Yaskawa INFORM job: R1_W35-36-A2(90,0)KM-OK.JBI

/JOB
//NAME R1_W35-36-A2(90,0)KM-OK
///FOLDERNAME KRIS-SCIANA
//POS
///NPOS 106,106,0,8,0,0
///TOOL 0
///POSTYPE PULSE
///PULSE
C00000=133203,-151163,-123299,-9717,62642,66340
C00001=174797,-117356,-116748,-21269,45538,71767
C00002=167772,-84002,-97078,-14094,48870,67877
C00003=165686,-78458,-91681,-12461,48082,67072
C00004=164380,-75033,-87353,-11529,47009,66627
C00005=163956,-73698,-86723,-11111,47244,66408
C00006=164380,-75033,-87353,-11529,47009,66627
C00007=164380,-75168,-86749,-11611,46576,66681
C00008=164380,-75033,-87353,-11529,47009,66627
C00009=153920,-88304,-92067,12036,39705,58111
C00010=154679,-95974,-98045,11331,39340,58456
C00011=173550,-85466,-94205,-27435,46132,79851
C00012=171230,-80075,-88912,-25751,44973,79042
C00013=169766,-76569,-85027,-24769,44003,78586
C00014=169296,-75333,-84452,-24248,44125,78311
C00015=169766,-76569,-85027,-24769,44003,78586
C00016=169766,-76625,-84526,-24915,43697,78678
C00017=169766,-76569,-85027,-24769,44003,78586
C00018=181492,-65329,-82160,-40061,58474,82712
C00019=194013,-96570,-98942,-47807,60580,87756
C00020=194013,-96570,-98942,-47807,60580,-51245
C00021=203995,-38561,-98383,-32392,87811,-61268
C00022=215531,-14026,-76080,-16989,89427,-64069
C00023=220381,23081,-47382,-28420,104834,-69323
C00024=222470,49341,-20749,-34117,110874,-70142
C00025=221806,39036,-18377,-32558,104968,-68512
C00026=221724,38193,-19154,-32548,104980,-68545
C00027=221793,39711,-18991,-32681,105579,-68702
C00028=221571,37477,-21115,-32657,105643,-68801
C00029=221571,37188,-20943,-32612,105427,-68735
C00030=222926,39369,-21029,-33153,106861,-68698
C00031=223966,38557,-20553,-33262,106600,-68250
C00032=226583,52363,-1545,-40953,111419,-72507
C00033=222365,54755,1299,-40199,109281,-73389
C00034=223739,53056,-5101,-41284,112199,-74042
C00035=218620,27349,-37181,-28911,103712,-69795
C00036=215610,8993,-54476,-21168,96493,-66602
C00037=215610,8993,-54476,-21168,96493,-66602
C00038=181695,45814,-29997,-12378,123903,-78661
C00039=175710,42579,-26967,-11179,119789,-80079
C00040=175710,41251,-26577,-11066,118883,-79984
C00041=175710,40643,-26381,-11016,118459,-79940
C00042=175710,41109,-26532,-11055,118786,-79974
C00043=179718,49925,-16862,-11334,117833,-78596
C00044=179718,48988,-16533,-11255,117161,-78526
C00045=179840,47754,-17901,-11295,117380,-78511
C00046=180929,51970,-15477,-11489,118166,-78244
C00047=186701,44441,-23841,-12245,120091,-76601
C00048=186701,44089,-23732,-12211,119848,-76573
C00049=186701,43441,-23524,-12148,119396,-76521
C00050=186701,43791,-23639,-12182,119641,-76549
C00051=186455,51365,-15254,-11993,118371,-76483
C00052=186455,50629,-14996,-11926,117845,-76424
C00053=186489,49492,-16087,-11940,117934,-76422
C00054=186464,52211,-15044,-12032,118669,-76513
C00055=197498,49366,-18518,-13101,120698,-73153
C00056=197498,48966,-18393,-13058,120422,-73119
C00057=197498,48360,-18192,-12995,119997,-73065
C00058=197498,48957,-18389,-13057,120414,-73118
C00059=196870,57395,-8813,-12787,118814,-73130
C00060=196870,56102,-8342,-12659,117882,-73019
C00061=196979,54648,-10005,-12704,118165,-73017
C00062=197536,59091,-8206,-12907,119386,-72980
C00063=207821,58971,-8346,-13607,120773,-69731
C00064=207821,58374,-8156,-13541,120362,-69677
C00065=207821,57623,-7899,-13459,119832,-69608
C00066=207821,58153,-8083,-13517,120207,-69656
C00067=206745,66427,1648,-13203,118369,-69786
C00068=206745,65417,2036,-13100,117629,-69695
C00069=206913,64191,584,-13146,117909,-69674
C00070=207056,66191,1124,-13250,118607,-69712
C00071=206807,76962,-1437,-14356,125245,-70692
C00072=178606,-7084,-71070,-5513,93657,-76211
C00073=178606,-12434,-69077,-5488,89699,-76039
C00074=178606,-14822,-67880,-5486,87744,-75953
C00075=166292,-14208,-67445,-208,87128,-79433
C00076=169556,-31327,-73894,-6745,74234,-79609
C00077=174833,-45592,-87827,-10016,75291,-78208
C00078=186297,-11008,-70403,4453,90875,-67936
C00079=188919,-9021,-66869,3281,89626,-67272
C00080=188904,-12076,-65397,3288,87157,-67339
C00081=208785,1057,-55100,-5592,87804,-61823
C00082=208466,4683,-57667,-5460,91212,-62059
C00083=165581,-6998,-67341,13530,92866,-73359
C00084=173591,4611,-59645,1891,100899,-73578
C00085=173591,2327,-58796,1879,99203,-73603
C00086=194456,6891,-54971,-5453,99565,-67936
C00087=194382,12631,-57077,-5530,103787,-68146
C00088=175852,-51384,-92394,-10580,75239,-77894
C00089=192163,-96959,-104003,-46570,61456,86648
C00090=152921,-122541,-108068,855,30408,65915
C00091=145454,-97772,-94010,9448,34954,61648
C00092=146863,-93018,-91491,7663,35693,62543
C00093=145492,-97786,-92846,9577,34237,61575
C00094=144929,-94903,-92971,9846,35841,61460
C00095=146748,-90810,-92138,6152,39176,62647
C00096=145438,-91687,-92725,7508,39198,61958
C00097=146922,-92489,-91306,7569,35844,62592
C00098=145432,-97676,-94179,9438,35110,61655
C00099=146808,-105604,-100046,7956,34504,62387
C00100=157428,-158903,-123496,-7044,21383,69853
C00101=121608,-159131,-116680,-7067,21310,69864
C00102=121608,-159131,-116680,-7067,21310,69864
C00103=6794,-159131,-116680,-7067,21310,69864
C00104=-19798,29541,-22378,6716,72357,-39538
C00105=-2234,110189,19387,12809,93315,-86753
BC00000=338018,1185852,1068216
BC00001=322204,1189606,1068222
BC00002=322204,1189606,1068222
BC00003=322204,1189606,1068222
BC00004=322204,1189606,1068222
BC00005=322204,1189606,1068222
BC00006=322204,1189606,1068222
BC00007=322204,1189606,1068222
BC00008=322204,1189606,1068222
BC00009=322204,1189606,1068222
BC00010=322204,1189606,1068222
BC00011=359570,1189606,1068222
BC00012=359570,1189606,1068222
BC00013=359570,1189606,1068222
BC00014=359570,1189606,1068222
BC00015=359570,1189606,1068222
BC00016=359570,1189606,1068222
BC00017=359570,1189606,1068222
BC00018=359570,1189606,1068222
BC00019=359570,1189606,1068222
BC00020=359570,1189606,1068222
BC00021=359570,1189606,1068222
BC00022=359570,1189606,1068222
BC00023=359570,1189606,1068222
BC00024=359570,1189606,1068222
BC00025=359570,1384690,1084352
BC00026=359570,1384690,1084352
BC00027=359570,1384690,1084352
BC00028=359570,1384690,1084352
BC00029=359570,1384690,1084352
BC00030=359570,1384690,1084352
BC00031=359570,1384690,1084352
BC00032=359570,1384690,1084352
BC00033=359570,1384690,1084352
BC00034=359570,1384690,1084352
BC00035=359570,1189606,1068222
BC00036=359570,1189606,1068222
BC00037=359570,1189606,1068222
BC00038=359570,1189606,1068222
BC00039=359570,1189606,1068222
BC00040=359570,1189606,1068222
BC00041=359570,1189606,1068222
BC00042=359570,1189606,1068222
BC00043=359570,1189606,1068222
BC00044=359570,1189606,1068222
BC00045=359570,1189606,1068222
BC00046=359570,1189606,1068222
BC00047=359570,1189606,1068222
BC00048=359570,1189606,1068222
BC00049=359570,1189606,1068222
BC00050=359570,1189606,1068222
BC00051=359570,1189606,1068222
BC00052=359570,1189606,1068222
BC00053=359570,1189606,1068222
BC00054=359570,1189606,1068222
BC00055=359570,1189606,1068222
BC00056=359570,1189606,1068222
BC00057=359570,1189606,1068222
BC00058=359570,1189606,1068222
BC00059=359570,1189606,1068222
BC00060=359570,1189606,1068222
BC00061=359570,1189606,1068222
BC00062=359570,1189606,1068222
BC00063=359570,1189606,1068222
BC00064=359570,1189606,1068222
BC00065=359570,1189606,1068222
BC00066=359570,1189606,1068222
BC00067=359570,1189606,1068222
BC00068=359570,1189606,1068222
BC00069=359570,1189606,1068222
BC00070=359570,1189606,1068222
BC00071=359570,1189606,1068222
BC00072=359570,1189606,1068222
BC00073=359570,1189606,1068222
BC00074=359570,1189606,1068222
BC00075=359570,1189606,1068222
BC00076=359570,1189606,1068222
BC00077=359570,1189606,1068222
BC00078=359570,1189606,1068222
BC00079=359570,1189606,1068222
BC00080=359570,1189606,1068222
BC00081=359570,1189606,1068222
BC00082=359570,1189606,1068222
BC00083=359570,1189606,1068222
BC00084=359570,1189606,1068222
BC00085=359570,1189606,1068222
BC00086=359570,1189606,1068222
BC00087=359570,1189606,1068222
BC00088=359570,1189606,1068222
BC00089=359570,1189606,1068222
BC00090=340811,1189606,1068222
BC00091=340087,1189606,1068222
BC00092=339797,1189606,1068222
BC00093=339797,1189606,1068222
BC00094=339797,1189606,1068222
BC00095=305385,1189606,1068222
BC00096=302058,1189606,1068222
BC00097=290425,1189606,1068222
BC00098=290715,1189606,1068222
BC00099=291439,1189606,1068222
BC00100=291439,1189606,1068222
BC00101=291439,1189606,1068222
BC00102=387760,1226770,1068222
BC00103=387760,1189606,1068222
BC00104=204934,1269644,1068209
BC00105=126121,1277269,1068204
///POSTYPE BASE
///RECTAN
///RCONF 0,0,0,0,0,0,0,0,0,0,0,0,0,0,0,0,0,0,0,0,0,0,0,0
P00006=0.222,-3.123,-1.508,0.0000,0.0000,0.0000
P00021=-0.225,-6.128,-0.405,0.0000,0.0000,0.0000
P00022=0.222,-3.123,-1.508,0.0000,0.0000,0.0000
P00025=-2.003,0.006,0.728,0.0000,0.0000,0.0000
P00030=5.926,-4.294,-1.390,0.0000,0.0000,0.0000
P00031=1.853,-0.001,-1.549,0.0000,0.0000,0.0000
P00032=1.957,0.503,-7.217,0.0000,0.0000,0.0000
///RCONF 0,0,0,0,1,0,0,0,0,0,0,0,0,0,0,0,0,0,0,0,0,0,0,0
P00033=-0.123,0.612,-5.012,0.0000,0.0000,0.0000
//INST
///DATE 2024/07/22 18:40
///ATTR SC,RW
///GROUP1 RB1,BS1
NOP
'r1_W35-36-A2(90,0)
'Path S1033 (for W914)
SFTOF
MOVJ C00000 BC00000 VJ=20.00
MOVJ C00001 BC00001 VJ=20.00
MOVL C00002 BC00002 V=166.7
MOVL C00003 BC00003 V=166.7
MOVL C00004 BC00004 V=60.0
REFP 3 C00005 BC00005
CALL JOB:SEARCH-R1
SET P021 P006
SFTON P021
MOVL C00006 BC00006 V=60.0
REFP 3 C00007 BC00007
CALL JOB:SEARCH-R1
SET P021 P006
SFTON P021
MOVL C00008 BC00008 V=60.0
MOVL C00009 BC00009 V=166.7
MOVL C00010 BC00010 V=166.7
'Path S1034 (for W914)
SFTOF
MOVL C00011 BC00011 V=166.7
MOVL C00012 BC00012 V=166.7
MOVL C00013 BC00013 V=60.0
REFP 3 C00014 BC00014
CALL JOB:SEARCH-R1
SET P022 P006
SFTON P022
MOVL C00015 BC00015 V=60.0
REFP 3 C00016 BC00016
CALL JOB:SEARCH-R1
SET P022 P006
SFTON P022
MOVL C00017 BC00017 V=60.0
MOVL C00018 BC00018 V=166.7
MOVJ C00019 BC00019 VJ=20.00
MOVJ C00020 BC00020 VJ=100.00
MOVJ C00021 BC00021 VJ=100.00
SFTOF
MOVJ C00022 BC00022 VJ=100.00
MOVJ C00023 BC00023 VJ=50.00
MOVJ C00024 BC00024 VJ=60.00
COMM PAUSE
COMM MOVL C00025 BC00025 V=60.0
COMM REFP 3 C00026 BC00026
COMM CALL JOB:SEARCH-R1
COMM SET P025 P006
COMM SFTON P025
COMM MOVL C00027 BC00027 V=83.3
COMM MOVL C00028 BC00028 V=60.0
COMM REFP 3 C00029 BC00029
COMM CALL JOB:SEARCH-R1
COMM SET P025 P006
COMM SFTON P025
COMM MOVL C00030 BC00030 V=60.0
COMM MOVL C00031 BC00031 V=166.7
COMM MACRO1 MJ#(0) ARGF6
COMM SFTON P025
COMM MOVJ C00032 BC00032 VJ=10.00
COMM MOVL C00033 BC00033 V=13.3
COMM ARCOF
COMM MOVL C00034 BC00034 V=83.3
COMM SFTOF
COMM PAUSE
MOVL C00035 BC00035 V=166.7
MOVJ C00036 BC00036 VJ=20.00
MOVL C00037 BC00037 V=166.7
MOVJ C00038 BC00038 VJ=20.00
MOVL C00039 BC00039 V=233.3
MOVL C00040 BC00040 V=60.0
REFP 3 C00041 BC00041
CALL JOB:SEARCH-R1
SET P030 P006
SFTON P030
MOVL C00042 BC00042 V=60.0
MOVL C00043 BC00043 V=100.0
MOVL C00044 BC00044 V=60.0
REFP 3 C00045 BC00045
CALL JOB:SEARCH-R1
SET P030 P006
SFTON P030
MOVL C00046 BC00046 V=60.0
SFTOF
MOVL C00047 BC00047 V=233.3
MOVL C00048 BC00048 V=60.0
REFP 3 C00049 BC00049
CALL JOB:SEARCH-R1
SET P031 P006
SFTON P031
MOVL C00050 BC00050 V=60.0
MOVL C00051 BC00051 V=100.0
MOVL C00052 BC00052 V=60.0
REFP 3 C00053 BC00053
CALL JOB:SEARCH-R1
SET P031 P006
SFTON P031
MOVL C00054 BC00054 V=60.0
SFTOF
MOVL C00055 BC00055 V=233.3
MOVL C00056 BC00056 V=60.0
REFP 3 C00057 BC00057
CALL JOB:SEARCH-R1
SET P032 P006
SFTON P032
MOVL C00058 BC00058 V=60.0
MOVL C00059 BC00059 V=100.0
MOVL C00060 BC00060 V=60.0
REFP 3 C00061 BC00061
CALL JOB:SEARCH-R1
SET P032 P006
SFTON P032
MOVL C00062 BC00062 V=60.0
SFTOF
MOVL C00063 BC00063 V=233.3
MOVL C00064 BC00064 V=60.0
REFP 3 C00065 BC00065
CALL JOB:SEARCH-R1
SET P033 P006
SFTON P033
MOVL C00066 BC00066 V=60.0
MOVL C00067 BC00067 V=100.0
MOVL C00068 BC00068 V=60.0
REFP 3 C00069 BC00069
CALL JOB:SEARCH-R1
SET P033 P006
SFTON P033
MOVL C00070 BC00070 V=60.0
SFTOF
MOVL C00071 BC00071 V=333.3
MOVL C00072 BC00072 V=333.3
MOVJ C00073 BC00073 VJ=15.00
SFTON P031
MOVL C00074 BC00074 V=100.0 PL=0
MACRO1 MJ#(0) ARGF9
ARCON
SFTON P030
MOVL C00075 BC00075 V=13.3
MOVL C00076 BC00076 V=13.3
ARCOF
MOVL C00077 BC00077 V=166.7
SFTOF
MOVJ C00078 BC00078 VJ=20.00
MOVJ C00079 BC00079 VJ=20.00
SFTON P032
MOVL C00080 BC00080 V=100.0 PL=0
ARCON
SFTON P033
MOVL C00081 BC00081 V=13.3
ARCOF
MOVJ C00082 BC00082 VJ=20.00
SFTOF
MOVJ C00083 BC00083 VJ=50.00
MOVJ C00084 BC00084 VJ=20.00
SFTON P031
MOVL C00085 BC00085 V=100.0 PL=0
ARCON
SFTON P032
MOVL C00086 BC00086 V=13.3
ARCOF
MOVJ C00087 BC00087 VJ=20.00
MOVJ C00088 BC00088 VJ=20.00
MOVJ C00089 BC00089 VJ=50.00
SFTOF
SFTON P022
MOVJ C00090 BC00090 VJ=20.00
MOVJ C00091 BC00091 VJ=20.00
MOVL C00092 BC00092 V=100.0 PL=0
REFP 1 C00093 BC00093
REFP 2 C00094 BC00094
MACRO1 MJ#(0) ARGF7
ARCON
MOVL C00095 BC00095 V=7.5
SFTON P021
MOVL C00096 BC00096 V=7.5
MOVL C00097 BC00097 V=7.5
ARCOF
MOVL C00098 BC00098 V=166.7
MOVL C00099 BC00099 V=166.7
SFTOF
MOVJ C00100 BC00100 VJ=100.00
MOVJ C00101 BC00101 VJ=60.00
MOVJ C00102 BC00102 VJ=100.00
MOVJ C00103 BC00103 VJ=100.00
MOVJ C00104 BC00104 VJ=100.00
MOVJ C00105 BC00105 VJ=100.00
END
